(* IEC 61131-3 sources: standardizer-tutorial-lib/src/ReceipeManager, 6 files *)

(* ---- IExecutables.st ---- *)
NAMESPACE Simatic.Ax.Tutorial
    INTERFACE IExecutable
        METHOD Execute END_METHOD
        METHOD HasFinished : BOOL END_METHOD
        METHOD GetState : StepState
        END_METHOD
        METHOD SetState
            VAR_INPUT
                state : StepState;
            END_VAR
        END_METHOD
        METHOD GetName : STRING
        END_METHOD
    END_INTERFACE

    TYPE
        StepState : (Idle, Busy, Done, Error) := Idle;
    END_TYPE
END_NAMESPACE

(* ---- IReceipeStep.st ---- *)
NAMESPACE Simatic.Ax.Tutorial
    // INTERFACE IStep
    //     METHOD GetName : STRING
    //     END_METHOD
    // END_INTERFACE

    TYPE
        ReceipeStepState : (Idle, Active, Done) := Idle;
    END_TYPE
END_NAMESPACE

(* ---- Runner.st ---- *)
USING Siemens.Ax.Collections;
NAMESPACE Simatic.Ax.Tutorial

    /// <summary>
    /// Class for running an instruction set
    /// </summary>
    CLASS PUBLIC Runner

        VAR PRIVATE
            _receipe : IReceipe;
            _currentListItem : IListItem;

            _currentStep : IExecutable;
            _state : RunnerState;
            _currentStateName : STRING;
        END_VAR

        METHOD PUBLIC LoadReceipe
            VAR_INPUT
                receipe : IReceipe;
            END_VAR

            _receipe := receipe;
            IF (_receipe = NULL) THEN
                _state := RunnerState#NoReceipeLoaded;
                RETURN;
            END_IF;

            _receipe.Init();
            _currentListItem := receipe.GetSteps().Tail();
            _currentStep ?= _currentListItem;
            _currentStateName := _currentStep.GetName();
            IF (_currentStep <> NULL) THEN
                _state := RunnerState#Idle;
            ELSE
                _state := RunnerState#NoReceipeLoaded;
            END_IF;
        END_METHOD

        /// <summary>
        /// Triggers the instructions one after each other
        /// </summary>
        /// <RETURNs>Void</RETURNs>
        METHOD PUBLIC RunCyclic

            IF _currentStep = NULL THEN
                _state := RunnerState#Error;
                RETURN;
            END_IF;

            IF _currentStep.HasFinished() THEN
                _currentStep.SetState(StepState#Idle);
                // Get next element from list and check if it's of type IReceipeStep
                _currentListItem := _currentListItem.NextItem();

                _currentStep ?= _currentListItem;
                _currentStep ?= _currentStep;
                IF (_currentStep <> NULL) THEN
                    _currentStep.SetState(state := StepState#Busy);
                    _currentStateName := _currentStep.GetName();
                    _state := RunnerState#StepSwitchover;
                ELSE
                    _state := RunnerState#Finished;
                END_IF;
            ELSE
                _state := RunnerState#Running;
                _currentStep.Execute();
            END_IF;
        END_METHOD

        METHOD PUBLIC GetState : RunnerState
            GetState := _state;
        END_METHOD
    END_CLASS
    TYPE
        RunnerState : (Running, Idle, StepSwitchover, Finished, NoReceipeLoaded, Error) := NoReceipeLoaded;
    END_TYPE

END_NAMESPACE

(* ---- IReceipe.st ---- *)
USING Siemens.Ax.Collections;

NAMESPACE Simatic.Ax.Tutorial
    INTERFACE IReceipe
        METHOD GetSteps : ILinkedList END_METHOD
        METHOD Init END_METHOD
    END_INTERFACE
END_NAMESPACE

(* ---- Receipe.st ---- *)
USING Siemens.Ax.Collections;

NAMESPACE Simatic.Ax.Tutorial
    CLASS ABSTRACT Receipe EXTENDS LinkedList IMPLEMENTS IReceipe

        // METHOD PUBLIC ABSTRACT Run : IStep END_METHOD

        METHOD PUBLIC ABSTRACT Init END_METHOD

        METHOD PUBLIC GetSteps : ILinkedList
            GetSteps := THIS;
        END_METHOD
END_CLASS
END_NAMESPACE

(* ---- ReceipeStep.st ---- *)
USING  Siemens.Ax.Collections;

NAMESPACE Simatic.Ax.Tutorial
    CLASS ABSTRACT ReceipeStep EXTENDS ListItem IMPLEMENTS IExecutable
        VAR PUBLIC
            Name : STRING := 'default value';
        END_VAR

        VAR PROTECTED
            _state : StepState;
        END_VAR

        METHOD PUBLIC HasFinished : BOOL
            HasFinished := _state = StepState#Done;
        END_METHOD

        METHOD PUBLIC ABSTRACT Execute END_METHOD

        METHOD PUBLIC GetState : StepState
            GetState := _state;
        END_METHOD

        METHOD PUBLIC SetState
            VAR_INPUT
                state : StepState;
            END_VAR
            _state := state;
        END_METHOD

        METHOD PUBLIC GetName : STRING
            GetName := Name;
        END_METHOD

    END_CLASS
END_NAMESPACE
